FUNCTION_BLOCK Luggage (* Composite Function Block Type *)
  (* Standard: 61499-2 *)
  (* Version 0.0, 5/29/2016, Andrei, nxtControl GmbH, template *)
  PACKAGE Main;
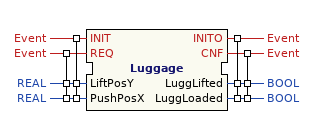
  EVENT_INPUT
    INIT WITH LiftPosY, PushPosX; (* Initialization Request *)
    REQ WITH LiftPosY, PushPosX; (* Normal Execution Request *)
  END_EVENT
  EVENT_OUTPUT
    INITO WITH LuggLifted, LuggLoaded; (* Initialization Confirm *)
    CNF WITH LuggLifted, LuggLoaded; (* Execution Confirmation *)
  END_EVENT
  VAR_INPUT
    LiftPosY : REAL;
    PushPosX : REAL;
  END_VAR
  VAR_OUTPUT
    LuggLifted : BOOL;
    LuggLoaded : BOOL;
  END_VAR
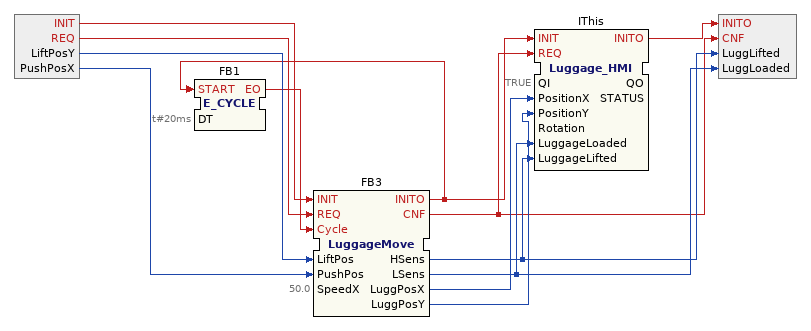
  FBS
    IThis : Luggage_HMI(QI := TRUE);
    FB1 : E_CYCLE(DT := t#20ms);
    FB3 : LuggageMove(SpeedX := 50.0);
  END_FBS
  EVENT_CONNECTIONS
    INIT TO FB3.INIT;
    REQ TO FB3.REQ;
    FB1.EO TO FB3.Cycle;
    FB3.INITO TO FB1.START;
    FB3.CNF TO CNF;
    FB3.INITO TO IThis.INIT;
    FB3.CNF TO IThis.REQ;
    IThis.INITO TO INITO;
  END_CONNECTIONS
  DATA_CONNECTIONS
    LiftPosY TO FB3.LiftPos;
    PushPosX TO FB3.PushPos;
    FB3.HSens TO LuggLifted;
    FB3.LSens TO LuggLoaded;
    FB3.LuggPosX TO IThis.PositionX;
    FB3.LuggPosY TO IThis.PositionY;
    FB3.LSens TO IThis.LuggageLoaded;
    FB3.HSens TO IThis.LuggageLifted;
  END_CONNECTIONS
END_FUNCTION_BLOCK
